PROGRAM PRG_Main_Report
VAR
	fbFormat   		  : FB_FormatString;
END_VAR

PRG_JsonWriter();
PRG_CurrentUserListWriter();
PRG_MethodReportWriter();
PRG_PostRunReportWriter();
PRG_PumpCalibrationReport();
PRG_UserHistoryReportWriter();
PRG_CreateJsonFile();
PRG_ReadJsonFile();

fbFormat(sFormat := 'Content/UI/PDFs/%s', arg1:= F_STRING(in:= GVL_Report.testPath), sOut => GVL_Report.localPDF);
WritingReportsHeads();

ACTION WritingReportsHeads:

GVL_Report.stReportHead.reportName:= 'TEGAN 1063 - Automated Sample Recovery System';
GVL_Report.stReportHead.databaseName:= 'Add a variable';
GVL_Report.stReportHead.printedBy:= 'printedby';
GVL_Report.stReportHead.reportDate:= 'putSystemVariable';
GVL_Report.stReportHead.systemID:= '???';
GVL_Report.stReportHead.page:= 'Create a page var';
END_ACTION

END_PROGRAM

(* stored: Version 1.1.0.1, ProductVersion 3.1.4024.12
   POU PRG_Main_Report: Id {aca5d804-13c7-4e2a-bb47-47660a1d3584}, SpecialFunc None
   Action WritingReportsHeads: Id {61f1259d-59bb-476a-8d99-722b62b89136} *)
